SUBAPPLICATION AuxInput_Dom_UP (* Subapplication Type *)
  (* Standard: 61499-2 *)
  (* Version 1.0, 2023-02-06, franz *)
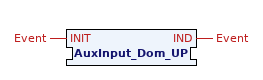
  EVENT_INPUT
    INIT;
  END_EVENT
  EVENT_OUTPUT
    IND;
  END_EVENT
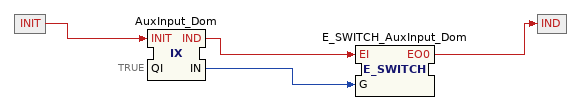
  FBS
    E_SWITCH_AuxInput_Dom : E_SWITCH;
    AuxInput_Dom : IX(QI := TRUE);
  END_FBS
  EVENT_CONNECTIONS
    AuxInput_Dom.IND TO E_SWITCH_AuxInput_Dom.EI;
    INIT TO AuxInput_Dom.INIT;
    E_SWITCH_AuxInput_Dom.EO0 TO IND;
  END_CONNECTIONS
  DATA_CONNECTIONS
    AuxInput_Dom.IN TO E_SWITCH_AuxInput_Dom.G;
  END_CONNECTIONS
END_SUBAPPLICATION
